INTERFACE I_Dimmable

METHOD GetLevel : BYTE
VAR_INPUT
END_VAR
END_METHOD

METHOD SetLevel : BOOL
VAR_INPUT
	// Level of dimmable
	Level: BYTE := 0;
END_VAR
END_METHOD

END_INTERFACE

(* stored: Version 1.1.0.1, ProductVersion 3.1.4024.5
   Itf I_Dimmable: Id {ec33756f-9a06-41e5-af2f-a28154902510}
   Method GetLevel: Id {db3bacc6-eef9-415f-9e7d-e9b2d36cd73b}
   Method SetLevel: Id {7d962b88-744b-449d-a149-4b7d4c39d8c9} *)
